//{attribute 'qualified_only'}
VAR_GLOBAL
	(* Gamma Ion Pump *)
	{attribute 'TcLinkTo' := 	'.q_xHVEna_DO	:=	TIIB[qRIXS_PLC_E2_EL2794]^Channel 1^Output;
								 .i_iPRESS		:=	TIIB[qRIXS_PLC_E3_EL3064]^AI Standard Channel 1^Value;
								 .i_xSP_DI		:=	TIIB[qRIXS_PLC_E1_EL1004]^Channel 1^Input
	'}
	{attribute 'pytmc' := '
		pv: QRIXS:OPT:PIP:01
		io: io
	'}
	qRIXS_OPT_PIP_01: FB_PIP_Gamma;
	
	(* Gamma Ion Pump *)
	{attribute 'TcLinkTo' := 	'.q_xHVEna_DO	:=	TIIB[qRIXS_PLC_E2_EL2794]^Channel 2^Output;
								 .i_iPRESS		:=	TIIB[qRIXS_PLC_E3_EL3064]^AI Standard Channel 2^Value;
								 .i_xSP_DI		:=	TIIB[qRIXS_PLC_E1_EL1004]^Channel 2^Input
	'}
	{attribute 'pytmc' := '
		pv: QRIXS:DET:PIP:01
		io: io
	'}
	qRIXS_DET_PIP_01: FB_PIP_Gamma;	
	
	
	(* -- Normally Closed Valve with Readback -- *)
	{attribute 'TcLinkTo' := 	'.i_xOpnLS	:=	TIIB[qRIXS_PNL1_E1_EL1004]^Channel 1^Input;
								 .i_xClsLS	:=	TIIB[qRIXS_PNL1_E1_EL1004]^Channel 2^Input;
								 .q_xOPN_DO	:=	TIIB[qRIXS_PNL1_E3_EL2004]^Channel 1^Output
	'}
	{attribute 'pytmc' := '
		pv: QRIXS:OPT:VGC:01
		io: io
	'}
	qRIXS_OPT_VGC_01: FB_VGC;
		
	{attribute 'TcLinkTo' := 	'.i_xOpnLS	:=	TIIB[qRIXS_PNL1_E1_EL1004]^Channel 3^Input;
								 .i_xClsLS	:=	TIIB[qRIXS_PNL1_E1_EL1004]^Channel 4^Input;
								 .q_xOPN_DO	:=	TIIB[qRIXS_PNL1_E3_EL2004]^Channel 2^Output
	'}
	{attribute 'pytmc' := '
		pv: QRIXS:BLW:VRC:01
		io: io
	'}
	qRIXS_BLW_VRC_01: FB_VRC;
	
	{attribute 'TcLinkTo' := 	'.i_xOpnLS	:=	TIIB[qRIXS_PNL1_E2_EL1004]^Channel 1^Input;
								 .i_xClsLS	:=	TIIB[qRIXS_PNL1_E2_EL1004]^Channel 2^Input;
								 .q_xOPN_DO	:=	TIIB[qRIXS_PNL1_E3_EL2004]^Channel 3^Output
	'}
	{attribute 'pytmc' := '
		pv: QRIXS:DET:VRC:01
		io: io
	'}
	qRIXS_DET_VRC_01: FB_VRC;
	
	
	(* MKS275 - Pirani *)
	{attribute 'TcLinkTo' := 	'.i_iPRESS_R	:=	TIIB[qRIXS_PNL1_E5_EL3174-0002]^AI Standard Channel 1^Value'}
	{attribute 'pytmc' := '
		pv: QRIXS:OPT:GPI:01
		io: io
	'}
	qRIXS_OPT_GPI_01: FB_MKS275;

	{attribute 'TcLinkTo' := 	'.i_iPRESS_R	:=	TIIB[qRIXS_PNL1_E5_EL3174-0002]^AI Standard Channel 2^Value'}
	{attribute 'pytmc' := '
		pv: QRIXS:DET:GPI:01
		io: io
	'}
	qRIXS_DET_GPI_01: FB_MKS275;
	
	
	(* MKS972 - Full range guage *)
	{attribute 'TcLinkTo' := 	'.i_iPRESS_R	:=	TIIB[qRIXS_PNL1_E5_EL3174-0002]^AI Standard Channel 3^Value'}
	{attribute 'pytmc' := '
		pv: QRIXS:BLW:GFR:01
		io: io
	'}
	qRIXS_BLW_GFR_01: FB_972;
	
	
	(* MKS500 - Cold cathode gauge *)
	{attribute 'TcLinkTo' := 	'.i_iPRESS_R		:=	TIIB[qRIXS_PNL1_E6_EL3174-0002]^AI Standard Channel 1^Value;
								 .i_xHV_ON			:=	TIIB[qRIXS_PNL1_E8_EL1124]^Channel 1^Input;
								 .i_xDisc_Active	:=	TIIB[qRIXS_PNL1_E8_EL1124]^Channel 2^Input;
								 .q_xHV_DIS			:=	TIIB[qRIXS_PNL1_E4_EL2624]^Channel 1^Output
	'}
	{attribute 'pytmc' := '
		pv: QRIXS:OPT:GCC:01
		io: io
	'}
	qRIXS_OPT_GCC_01: FB_MKS500;
	
	
	{attribute 'TcLinkTo' := 	'.i_iPRESS_R		:=	TIIB[qRIXS_PNL1_E6_EL3174-0002]^AI Standard Channel 2^Value;
								 .i_xHV_ON			:=	TIIB[qRIXS_PNL1_E8_EL1124]^Channel 3^Input;
								 .i_xDisc_Active	:=	TIIB[qRIXS_PNL1_E8_EL1124]^Channel 4^Input;
								 .q_xHV_DIS			:=	TIIB[qRIXS_PNL1_E4_EL2624]^Channel 2^Output
	'}
	{attribute 'pytmc' := '
		pv: QRIXS:DET:GCC:01
		io: io
	'}
	qRIXS_DET_GCC_01: FB_MKS500;
END_VAR

(* stored: Version 1.1.0.1, ProductVersion 3.1.4022.18
   GVL GVL_Devices: Id {94862fa7-5f8b-4725-b95d-44f5a97a24ca} *)
